PROGRAM Prg_WritePersistentVars
VAR
	//fb_FB_S_UPS: FB_S_UPS_CX51x0;
	fb_FB_S_UPS: FB_S_UPS_CX9020_U900;
	fb_FB_WritePersistentData: FB_WritePersistentData;
	
	_WritePersis: BOOL;
END_VAR

fb_FB_S_UPS(
		sNetID:='' , 
		iPLCPort:=851 , 
		//iplPort:= , 
		tTimeout:= , 
		eUpsMode:=eSUPS_WrPersistData_Shutdown , 
		ePersistentMode:=SPDM_2PASS , 
		tRecoverTime:= , 
		bPowerFailDetect=> , 
		eState=> );
		
		

fb_FB_WritePersistentData(
	NETID:= , 
	PORT:= 851, 
	START:=_WritePersis , 
	TMOUT:= , 
	MODE:= , 
	BUSY=> , 
	ERR=> , 
	ERRID=> );

END_PROGRAM

(* stored: Version 1.1.0.1, ProductVersion 3.1.4024.13
   POU Prg_WritePersistentVars: Id {3bc90efe-a9ce-4064-9b5c-f4509fe44ce9}, SpecialFunc None *)
